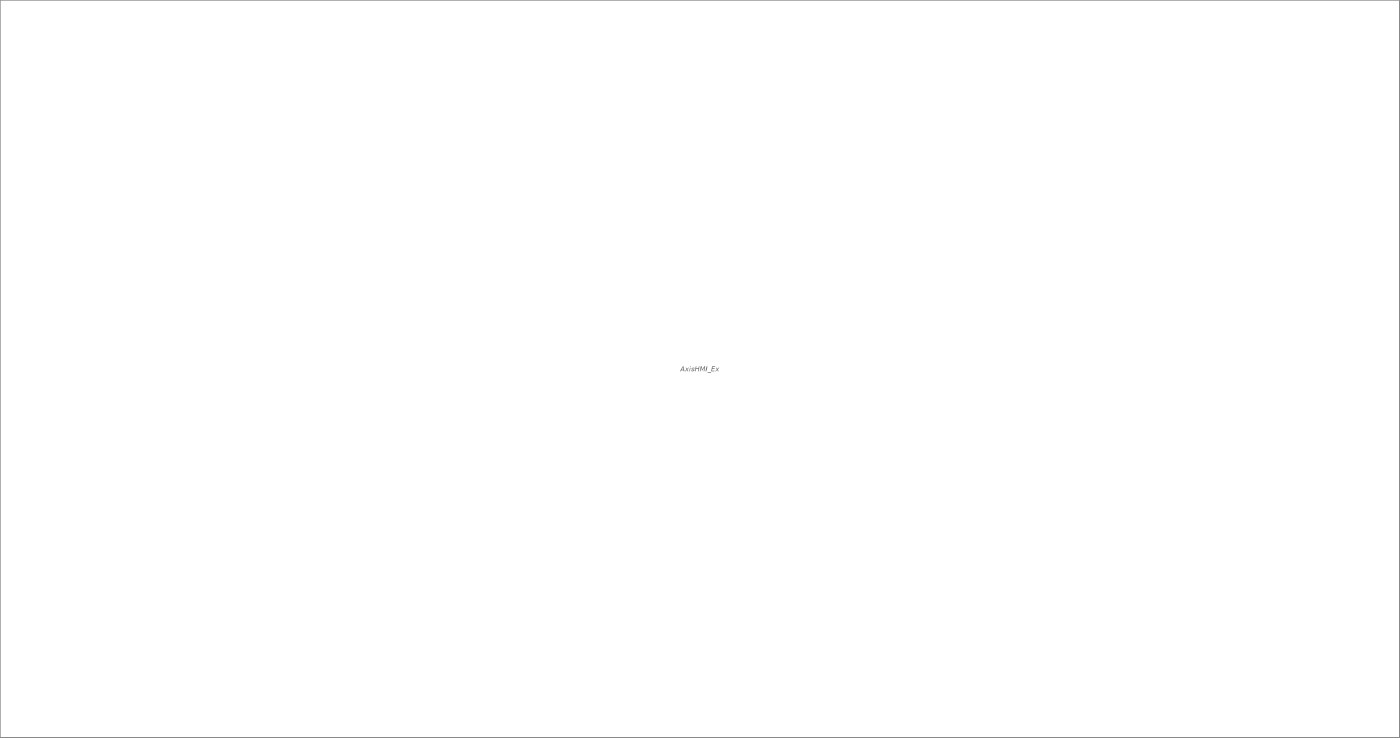
VISUALIZATION visu_PM  // 2048x1080
    TabControl (0,0 2048x1080)
        shows AxisHMI_Ex(stAxisHMI := GVL.pm[G_HMI.iPM].buffer[0].st_mcAxis, mcAxis := GVL.pm[G_HMI.iPM].buffer[0].mcAxis, xError := GVL.pm[G_HMI.iPM].buffer[0].mcAxis.xError)
        shows AxisHMI_Ex(stAxisHMI := GVL.pm[G_HMI.iPM].buffer[1].st_mcAxis, mcAxis := GVL.pm[G_HMI.iPM].buffer[1].mcAxis, xError := GVL.pm[G_HMI.iPM].buffer[1].mcAxis.xError)
        shows v_pm_0(dIO_PM := GVL.pm[G_HMI.iPM])
        shows Axis_HMI(st_axis_HMI := st_mcAxis[EN_Axis.Grip_axis])
        shows v_rem_1(dIO_ReM := GVL.pm[G_HMI.iModule])
        [0]: TabTitle=Buffer0
        [1]: TabTitle=Buffer1
        [6]: TabTitle=Gripper
        [2]: AxisHMI=gantrybase.st_mcAxis[EN_Axis.Z], mcAxis=gantrybase.mcAxis[EN_Axis.Z], Error=gantrybase.mcAxis[EN_Axis.Z].xError
        p699000190: gantrybase.st_mcAxis[EN_Axis.X]
        p2837713833: gantrybase.mcAxis[EN_Axis.Z].sAxisName
        p520277221: gantrybase.mcAxis[EN_Axis.X].xError
        p3331604638: gantrybase.st_mcAxis[EN_Axis.Z]
        p1813558639: gantrybase.mcAxis[EN_Axis.Z].xError
        p1563495665: gantrybase.st_mcAxis[EN_Axis.Y]
        p2070126892: gantrybase.mcAxis[EN_Axis.Y].xError
        p3435970784: gantrybase.mcAxis[EN_Axis.X]
        p2829954345: gantrybase.mcAxis[EN_Axis.Y]
        p3218520426: gantrybase.mcAxis[EN_Axis.Z]
END_VISUALIZATION

(* stored: Version 1.1.0.1, ProductVersion 3.1.4024.12
   Visu visu_PM: Id {54bce5ab-f9ca-42f8-8fb0-7aec53f0e7b9} *)
